FUNCTION_BLOCK SR (* Basic Function Block Type *)
  (* Standard: 61499-2 *)
  (* Version 0.0, 6/3/2016, Andrei, nxtControl GmbH, Template *)
  PACKAGE Main;
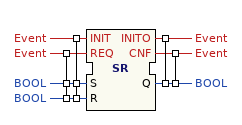
  EVENT_INPUT
    INIT WITH S, R; (* Initialization Request *)
    REQ WITH S, R; (* Normal Execution Request *)
  END_EVENT
  EVENT_OUTPUT
    INITO WITH Q; (* Initialization Confirm *)
    CNF WITH Q; (* Execution Confirmation *)
  END_EVENT
  VAR_INPUT
    S : BOOL; (* Input event qualifier *)
    R : BOOL;
  END_VAR
  VAR_OUTPUT
    Q : BOOL; (* Output event qualifier *)
  END_VAR
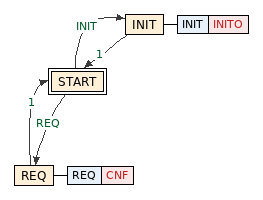
  EC_STATES
    START; (* Initial State *)
    INIT : INIT -> INITO; (* Initialization *)
    REQ : REQ -> CNF; (* Normal execution *)
  END_STATES
  EC_TRANSITIONS
    START TO INIT := INIT;
    INIT TO START := 1;
    START TO REQ := REQ;
    REQ TO START := 1;
  END_TRANSITIONS
  ALGORITHM INIT IN ST: (* Initialization algorithm *)
Q := FALSE;
  END_ALGORITHM
  ALGORITHM REQ IN ST: (* Normally executed algorithm *)
IF S AND NOT(R) THEN
	Q := TRUE;
ELSE
	Q := FALSE;
END_IF;
  END_ALGORITHM
END_FUNCTION_BLOCK
